(* Logix 5000 project; controller Modbus_TCP_Client_Example vendor 1 type 14 code 154 rev 32.15; software revision 32.05 *)

TASK Modbus_Task (periodic, rate 50 ms, priority 10, watchdog 500 ms) : Modbus_Program   // Conveyor MDXT

MODULES
   Local : vendor 1 type 14 code 154 (PointIO 0, rev 32.15)
      Discrete_IO : Embedded (PointIO 1, rev 32.11, Output RPI 20 ms)
END_MODULES

TYPE AMP_Alarm_Word :   // Applied Motion Input Assembly - Alarm Word
STRUCT
   Position_Limit : BOOL;   // Position Limit
   CCW_Limit : BOOL;   // CCW Limit
   CW_Limit : BOOL;   // CW Limit
   Over_Temp : BOOL;   // Over Temp
   Excess_Regen_or_Internal_Voltage : BOOL;   // Excess Regen or Internal Voltage
   Over_Voltage : BOOL;   // Over Voltage
   Under_Voltage : BOOL;   // Under Voltage
   Over_Current : BOOL;   // Over Current
   Open_Motor_Windings : BOOL;   // Open Motor Windings
   Bad_Encoder : BOOL;   // Bad Encoder
   Comm_Error : BOOL;   // Comm Error
   Bad_Flash : BOOL;   // Bad Flash
   No_Move : BOOL;   // No Move
   NA_1 : BOOL;   // NA 1
   Blank_Q_Segment : BOOL;   // Blank Q Segment
   NA_2 : BOOL;   // NA 2
END_STRUCT
END_TYPE

TYPE AMP_Input_Assembly_Servo_v2 :   // Applied Motion Servo Drive Input Assembly Version 1.0
STRUCT
   Control_Word_Received : DINT;   // Control Word Status equals to Control Words sent in Output Assembly
   OpCode1_Received : DINT;   // OpCode 1 Status equals to OpCode1 sent in Output Assembly
   Control_Mode : DINT;   // Control Mode Status: Position, Torque, Gear
   Status_Code : DINT;   // Status Code
   Alarm_Code : DINT;   // Alarm Code
   Supply_Voltage : DINT;   // Supply Voltage 0.1 V: ex. 242=24.2V
   Applied_Torque : DINT;   // Total Applied Torque %
   Drive_Temperature : DINT;   // Drive Temperature 0.1 deg C: ex. 305=30.5 C
   Encoder_Position : DINT;   // Encoder Position
   Second_Encoder_Position : DINT;   // Absolute Position
   Position_Error : DINT;   // Position Error in Counts
   Actual_Velocity_RPS : DINT;   // Actual Velocity rev/sec*2: ex. 480=2 rev/sec
   Digital_Outputs : DINT;   // Digital Output Status
   Digital_Inputs : DINT;   // Digital Input Status
   Analog_Output1 : DINT;   // 0 = min V, 16383 = max V
   Analog_Output2 : DINT;   // 0 = min V, 16383 = max V
   Analog_Input1 : DINT;   // 0 = min V, 16383 = max V
   Analog_Input2 : DINT;   // 0 = min V, 16383 = max V
   Torque_Limit : DINT;   // Torque Limit Set Point Feedback
   Second_Encoder_Speed : DINT;   // External Encoder Speed Feedback if any
END_STRUCT
END_TYPE

TYPE AMP_Input_Assembly_v2 :   // Applied Motion Drive Input Assembly Version 2.0
STRUCT
   Status_Code : DINT;   // Status Code
   Alarm_Code : DINT;   // Alarm Code
   Voltage : DINT;   // Supply Voltage (x0.1V)
   Current : DINT;   // Actual Current (mA)
   Temp : DINT;   // Drive Temperature (0.1 deg C)
   Encoder_Position : DINT;   // Encoder Position (20,000 counts = 1 shaft turn)
   Absolute_Position : DINT;   // Absolute Position (20,000 counts = 1 shaft turn)
   Position_Error : DINT;   // Position Error (counts)
   Actual_Velocity : DINT;   // Actual Velocity (rev/sec * 240, 0 when no encoder)
   Extended_Inputs : DINT;   // Input Status (Extended)
   Main_Board_Inputs : DINT;   // Input Status (Main board)
   Word11 : DINT;   // Reserved
   Analog_Input_1 : DINT;   // Analog Input 1 (ADC counts, 0=min V, 16383 = max V)
   Analog_Input_2 : DINT;   // Analog Input 2 (ADC counts, 0=min V, 16383 = max V)
END_STRUCT
END_TYPE

TYPE AMP_Status_Word :   // Applied Motion Input Assembly Status Word
STRUCT
   Enabled : BOOL;   // Motor Enabled (Motor Disabled if this bit = 0)
   Sampling : BOOL;   // Sampling (for Quick Tuner)
   Drive_Fault : BOOL;   // Drive Fault (check Alarm Code)
   In_Position : BOOL;   // In Position (motor is in position)
   Moving : BOOL;   // Moving (motor is moving)
   Jogging : BOOL;   // Jogging (currently in jog mode)
   Stopping : BOOL;   // Stopping (in the process of stopping from a stop command)
   Waiting : BOOL;   // Waiting (for an input; executing a WI command)
   Saving : BOOL;   // Saving (parameter data is being saved)
   Alarm_Present : BOOL;   // Alarm present (check Alarm Code)
   Homing : BOOL;   // Homing (executing an SH command)
   Wait_Time : BOOL;   // Waiting (for time; executing a WD or WT command)
   Wizard_Running : BOOL;   // Wizard running (Timing Wizard is running)
   Checking_Encoder : BOOL;   // Checking encoder (Timing Wizard is running)
   Q_Program_Running : BOOL;   // Q Program is running
   Initializing : BOOL;   // Initializing (happens at power up) ; Servo Ready (for SV200 drives only)
END_STRUCT
END_TYPE

TYPE AMP_Status_Word_Servo :   // Applied Motion Input Assembly Status Word 'SC'
STRUCT
   Enabled : BOOL;   // Motor Enabled (Motor Disabled if this bit = 0)
   Sampling : BOOL;   // Sampling
   Drive_Fault : BOOL;   // Drive Fault (check Alarm Code)
   In_Position : BOOL;   // In Position (motor is in position)
   Moving : BOOL;   // Moving (motor is moving)
   Jogging : BOOL;   // Jogging (currently in jog mode)
   Stopping : BOOL;   // Stopping (in the process of stopping from a stop command)
   Waiting : BOOL;   // Waiting (for an input; executing a WI command)
   Saving : BOOL;   // Saving (parameter data is being saved)
   Alarm_Present : BOOL;   // Alarm present (check Alarm Code)
   Homing : BOOL;   // Homing (executing an SH command)
   Wait_Time : BOOL;   // Waiting (for time; executing a WD or WT command)
   Wizard_Running : BOOL;   // Wizard running (Timing Wizard is running)
   Checking_Encoder : BOOL;   // Checking encoder (Timing Wizard is running)
   Q_Program_Running : BOOL;   // Q Program is running
   Servo_Ready : BOOL;   // Servo Ready;Initializing (happens at power up)
   CSP_Following : BOOL;
   In_Velocity : BOOL;   // Velocity Reached
   Zero_Speed : BOOL;   // Motor is standstill
   Torque_Reached : BOOL;   // Toruqe Target Reached
   In_Torque : BOOL;   // Current Control Mode is Torque
   Group2_PID : BOOL;   // The Second Set of Gain is Valid
   Secondary_Control_Mode : BOOL;   // Second Control Mode is in Operation
   Velocity_Reached : BOOL;   // Velocity Target Reached
   Homing_Complete : BOOL;   // Homing Completed Feedback
END_STRUCT
END_TYPE

TYPE raC_UDT_ModbusClientConnection :
STRUCT
   LocalSlot : SINT;   // Local Slot for Ethernet module. For ControlLogix - L8x, EN2T(R) - use the actual module slot. For CompactLogix use slot 0.
   LocalAddress : STR0016;   // Used only for controllers with more than 1 local IP address (5380, 5480). For all others must be blank.
   DestAddress : STR0016;   // The IP address for the Modbus TCP Slave device to connect to
   DestinationPort : DINT;   // Default Modbus is 502
   MSG_Src : SINT[500];   // Placeholder for message source
   MSG_Dest : SINT[500];   // Placeholder for message destination
END_STRUCT
END_TYPE

TYPE raC_UDT_ModbusClientData :
STRUCT
   Coils_0xxx : BOOL[1024];
   DiscInputs_1xxx : BOOL[1024];
   InpRegisters_3xxx : INT[1024];
   HoldRegisters_4xxx : INT[1024];
END_STRUCT
END_TYPE

TYPE raC_UDT_ModbusClientHMI :
STRUCT
   Parameters : raC_UDT_ModbusClientConnection;
   Transaction : raC_UDT_ModbusClientTransaction;
   Index0x : DINT;
   Index1x : DINT;
   Index3x : DINT;
   Index4x : DINT;
   DataValue : INT[65];
   DataAddr : DINT[65];
   TransactionIndex : DINT;
   RemoteAddrStart : DINT;
   RemoteAddrEnd : DINT;
   LocalAddrEnd : DINT;
END_STRUCT
END_TYPE

TYPE raC_UDT_ModbusClientTransaction :
STRUCT
   Enabled : BOOL;   // Enables (1) or disables (0) the transaction
   PollInterval : DINT;   // Time between triggers in milliseconds. Minimum is 80 msec. Anyting below 80 will be set to 1 seconds
   TransType : INT;   // Transaction code for the Modbus Protocol. Acceptable values are 1-Coil Read, 2- Discrete Input read, 3-Holding Register Read, 4-Input Register Read, 5-Write Single Coil, 6-Single Holding Register Write, 15-Multiple Coil Write, 16 Multiple Holding Register Write
   StationID : SINT;   // Station ID ( Unit Identifier). Commonly used if going through a gateway or bridge in which case it is the device address on the other side of the gateway. Other wise leave as 0
   BeginAddress : DINT;   // Beginning address in remote device to read from or write to.
   Count : INT;   // The number of items in remote device to read from or write to.
   LocalAddress : INT;   // Beginning address in in this programs' "_Data" arrays
   TransComplete : BOOL;   // Transaction Complete Flag. Check the TransStat to see if the transaction was successful or if a Modbus exception code was returned.
   TransStat : INT;   // Status result of the transaction. 0 = success, 1 = in process 2 = retry -1 = exception
   Diagnostic : raC_UDT_ModbusClientTransactionDiag;
END_STRUCT
END_TYPE

TYPE raC_UDT_ModbusClientTransactionDiag :
STRUCT
   Request : STR0500;   // Actual buffer used to build the modbus request that is transmited to the remote node.
   ReqBuilt : BOOL;   // Transaction request string is built, clear this if anything is changed in a read operation to rebuild the Request string.
   Overlap : BOOL;   // Transaction is not completing before next trigger
   Overload : BOOL;   // Transaction is not completing because of excessive Overlaps in one or more transactions
   TransID : INT;   // Serial Number of the actual Ethernet Transaction used to match to the appropriate Reply
   TransLastError : INT;   // Last Error on transaction. 0-Success, -2 Network write error, -3 Local write error, -4 Network Read Error, -5 Local Read Error, -6 Connection failed.. -12 Invalid Trans code, -13 Out of data array range.
   IntervalTimer : TIMER;   // IntervalTimer, used to trigger transaction
   NoReplyCounter : COUNTER;   // No Reply Counter
   PendingTimer : TIMER;   // Timing pending requests
END_STRUCT
END_TYPE

TYPE raC_UDT_ModbusConnectParam :   // Parameterss for the OpenConnection Service
STRUCT
   Timeout : DINT;
   DestAddr : STR0032;
END_STRUCT
END_TYPE

TYPE raC_UDT_ModbusCreateParam :
STRUCT
   Type : DINT;   // Type 1-TCP, 2-UDP
   Family : INT;   // Address Family Must be 2
   Port : INT;   // Local Port Number
   Addr : DINT;   // Local IP Address
END_STRUCT
END_TYPE

TYPE STR0008 :
STRUCT
   LEN : DINT;
   DATA : SINT[8];
END_STRUCT
END_TYPE

TYPE STR0016 :
STRUCT
   LEN : DINT;
   DATA : SINT[16];
END_STRUCT
END_TYPE

TYPE STR0032 :
STRUCT
   LEN : DINT;
   DATA : SINT[32];
END_STRUCT
END_TYPE

TYPE STR0500 :
STRUCT
   LEN : DINT;
   DATA : SINT[500];
END_STRUCT
END_TYPE

TYPE STR4096 :
STRUCT
   LEN : DINT;
   DATA : SINT[4096];
END_STRUCT
END_TYPE

ADD_ON_INSTRUCTION AMP_Absolute_Move   (* revision 1.0 *)
// Applied Motion - Absolute Move AOI
// Help:
// The Absolute Move AOI is used to move an axis to a specified absolute position.
VAR_IN_OUT
   Input : DINT[14]; {required}   // Drive Input Assembly
   Output : DINT[16]; {required}   // Drive Output Assembly
        [0]   // Command Word
        [10]   // Data/Register 1
        [11]   // Data/Register 2
        [1]   // Jog Speed (0.25 rev/min)
        [2]   // Jog Acceleration (10 rev/s/s)
        [3]   // Jog Deceleration (10 rev/s/s)
        [4]   // Point-to-Point Velocity (0.25 rev/min)
        [5]   // Point-to-Point Acceleration (10 rev/min/s)
        [6]   // Point-to-Point Deceleration (10 rev/min/s)
        [7]   // Point-to-Point Distance (Motor steps)
        [9]   // (2x ASCII Letters in 16 lower word)
END_VAR
VAR_INPUT
   RPI : DINT := 100; {visible}   // Drive Connection Request Packet Interval (milliseconds)
   Start : BOOL; {required}   // Start the Relative Move
   Position : DINT; {required}   // Destination Position (steps, negative = reverse)
   Speed : REAL; {required}   // Velocity of Move (rev/min)
   Acc : REAL; {required}   // Acceleration of Move (rev/s/s)
   Dec : REAL; {required}   // Deceleration (rev/s/s)
END_VAR
VAR_OUTPUT
   Sent : BOOL; {access Read Only, visible}   // Move has been sent to drive
   In_Progress : BOOL; {access Read Only, visible}   // Move in progress
   Done : BOOL; {access Read Only, visible}   // Move completed without errors - desired position reached
   Error : BOOL; {access Read Only, visible}   // Move failed to complete - drive not ready or faulted
   State : DINT := 10; {access Read Only}   // Internal state of progress
END_VAR
VAR
   Loc_StatusCode : AMP_Status_Word;
   Loc_CommandOff_Timer : TIMER;   // Timer to make sure command value was 0 before sending a new command
   Loc_CommandOn_Timer : TIMER;   // Timer to make sure command value is set long enough to be sent to drive
   Loc_Input_Assembly : AMP_Input_Assembly_v2; {access None}
   Loc_Start_ONS : BOOL; {access None}
   Loc_AlarmCode : AMP_Alarm_Word; {access None}
END_VAR

ROUTINE Logic   (* ladder *)
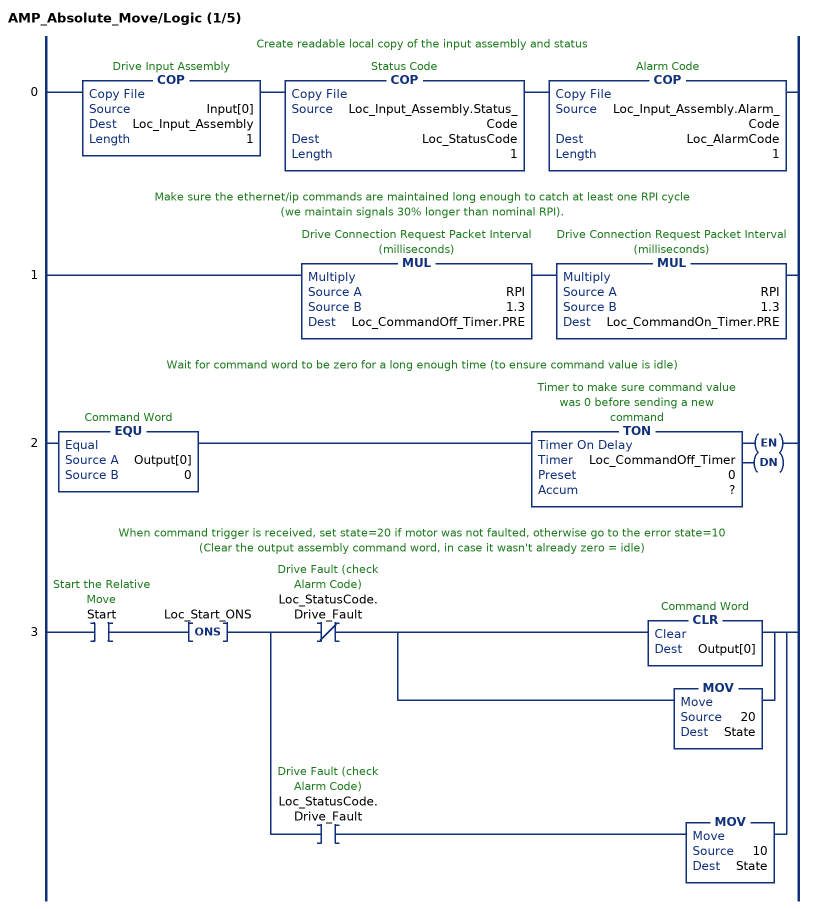
   // Create readable local copy of the input assembly and status
   0: COP(Input[0],Loc_Input_Assembly,1)COP(Loc_Input_Assembly.Status_Code,Loc_StatusCode,1)COP(Loc_Input_Assembly.Alarm_Code,Loc_AlarmCode,1);
   // Make sure the ethernet/ip commands are maintained long enough to catch at least one RPI cycle
   // (we maintain signals 30% longer than nominal RPI).
   1: MUL(RPI,1.3,Loc_CommandOff_Timer.PRE)MUL(RPI,1.3,Loc_CommandOn_Timer.PRE);
   // Wait for command word to be zero for a long enough time (to ensure command value is idle)
   2: EQU(Output[0],0)TON(Loc_CommandOff_Timer,?,?);
   // When command trigger is received, set state=20 if motor was not faulted, otherwise go to the error state=10
   // (Clear the output assembly command word, in case it wasn't already zero = idle)
   3: XIC(Start)ONS(Loc_Start_ONS)[XIO(Loc_StatusCode.Drive_Fault) [CLR(Output[0]) ,MOV(20,State) ] ,XIC(Loc_StatusCode.Drive_Fault) MOV(10,State) ];
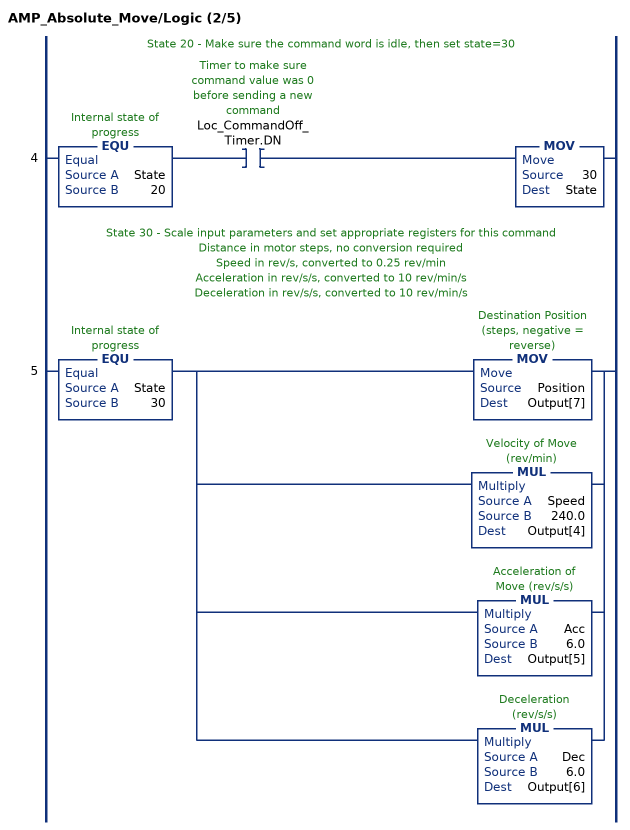
   // State 20 - Make sure the command word is idle, then set state=30
   4: EQU(State,20)XIC(Loc_CommandOff_Timer.DN)MOV(30,State);
   // State 30 - Scale input parameters and set appropriate registers for this command
   // Distance in motor steps, no conversion required
   // Speed in rev/s, converted to 0.25 rev/min
   // Acceleration in rev/s/s, converted to 10 rev/min/s
   // Deceleration in rev/s/s, converted to 10 rev/min/s
   5: EQU(State,30)[MOV(Position,Output[7]) ,MUL(Speed,240.0,Output[4]) ,MUL(Acc,6.0,Output[5]) ,MUL(Dec,6.0,Output[6]) ];
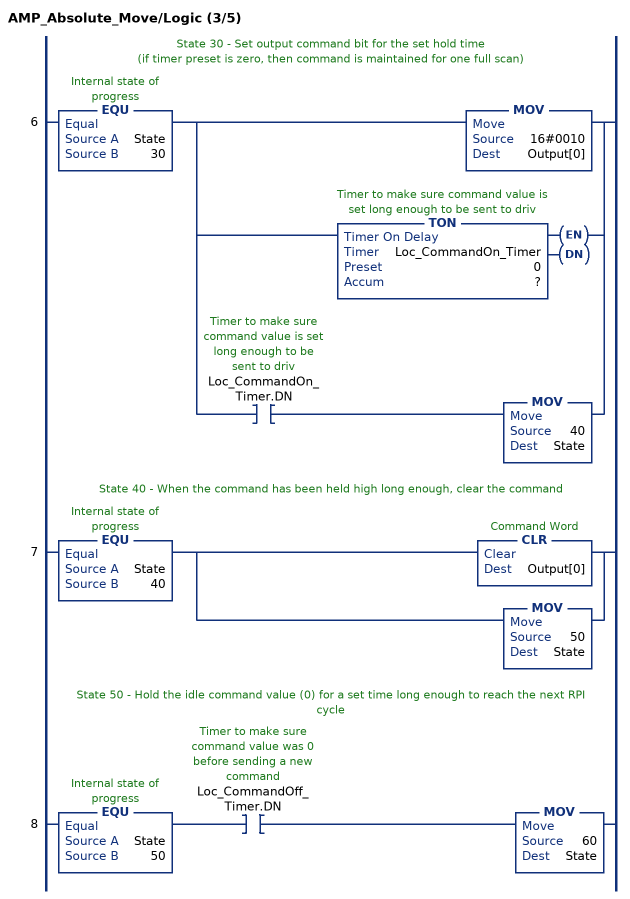
   // State 30 - Set output command bit for the set hold time
   // (if timer preset is zero, then command is maintained for one full scan)
   6: EQU(State,30)[MOV(16#0010,Output[0]) ,TON(Loc_CommandOn_Timer,?,?) ,XIC(Loc_CommandOn_Timer.DN) MOV(40,State) ];
   // State 40 - When the command has been held high long enough, clear the command
   7: EQU(State,40)[CLR(Output[0]) ,MOV(50,State) ];
   // State 50 - Hold the idle command value (0) for a set time long enough to reach the next RPI cycle
   8: EQU(State,50)XIC(Loc_CommandOff_Timer.DN)MOV(60,State);
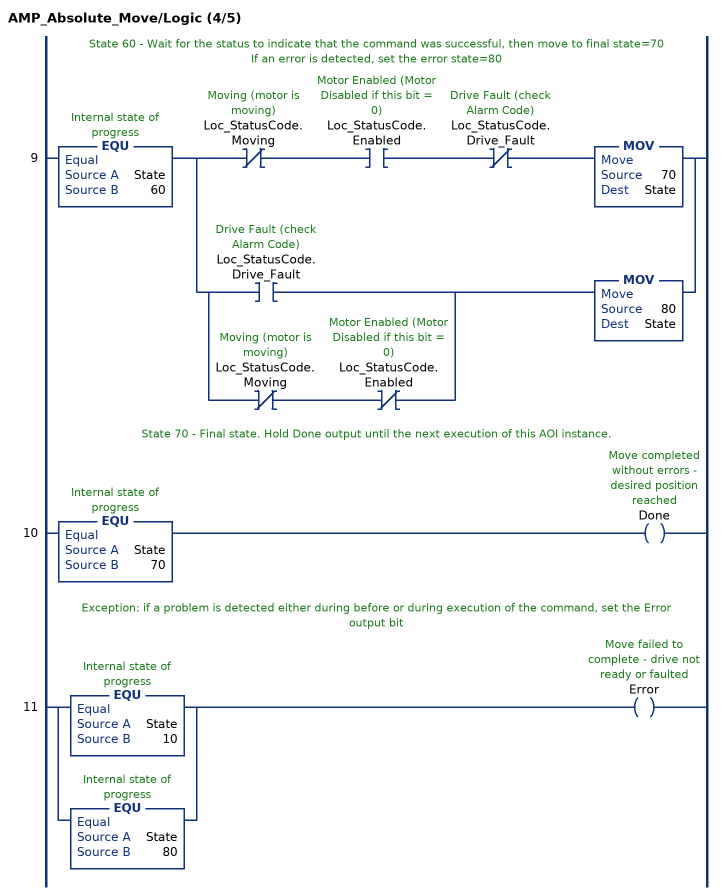
   // State 60 - Wait for the status to indicate that the command was successful, then move to final state=70
   // If an error is detected, set the error state=80
   9: EQU(State,60)[XIO(Loc_StatusCode.Moving) XIC(Loc_StatusCode.Enabled) XIO(Loc_StatusCode.Drive_Fault) MOV(70,State) ,[XIC(Loc_StatusCode.Drive_Fault) ,XIO(Loc_StatusCode.Moving) XIO(Loc_StatusCode.Enabled) ] MOV(80,State) ];
   // State 70 - Final state. Hold Done output until the next execution of this AOI instance.
   10: EQU(State,70)OTE(Done);
   // Exception: if a problem is detected either during before or during execution of the command, set the Error output bit
   11: [EQU(State,10) ,EQU(State,80) ]OTE(Error);
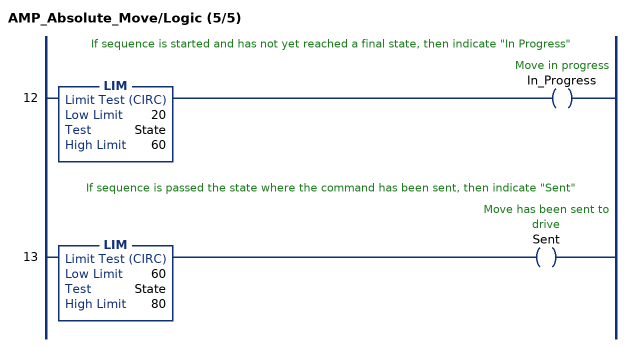
   // If sequence is started and has not yet reached a final state, then indicate "In Progress"
   12: LIM(20,State,60)OTE(In_Progress);
   // If sequence is passed the state where the command has been sent, then indicate "Sent"
   13: LIM(60,State,80)OTE(Sent);
END_ROUTINE
END_ADD_ON_INSTRUCTION

ADD_ON_INSTRUCTION AMP_Absolute_Move_Servo   (* revision 1.0, vendor Applied Motion Products Inc. *)
// Applied Motion - Motor Absolute Move - AOI
// Help:
// The Absolute Move AOI is used to move an axis to a specified absolute position(FP).
VAR_IN_OUT
   Input : DINT[20]; {required}   // Drive Input Assembly
        [16]   // Analog_Input1
        [4]   // Alarm_Code
        [0]   // Control_Word_Received
        [10]   // Position_Error
        [11]   // Actual_Velocity_RPS
        [12]   // Digital_Outputs
        [13]   // Digital_Inputs
        [14]   // Analog_Output1
        [15]   // Analog_Output2
        [17]   // Analog_Input2
        [18]   // Torque_Limit
        [19]   // Second_Encoder_Speed
        [1]   // OpCode1_Received
        [2]   // Control_Mode
        [3]   // Status_Code
        [5]   // Supply_Voltage
        [6]   // Applied_Torque
        [7]   // Drive_Temperature
        [8]   // Encoder_Position
        [9]   // Second_Encoder_Position
   Output : DINT[11]; {required}   // Drive Output Assembly
        [10]   // Reserved
        [4]   // Target Velocity
        [0]   // Control Word
        [3]   // Target Pos
        [1]   // OpCode 1
        [2]   // OpCode 2
        [5]   // Porifle Acceleration
        [6]   // Profile Deceleration
        [7]   // Target Torque
        [8]   // OpCode 3
        [9]   // OpCode 4
END_VAR
VAR_INPUT
   Start : BOOL; {required}   // Start the Absolute Move
   Position : DINT; {required}   // Destination Position (negative = reverse)
   Speed_rps : REAL; {required}   // Velocity of Move (rev/sec)
   Acc : REAL; {required}   // Acceleration of Move (rev/s/s)
   Dec : REAL; {required}   // Deceleration of Move (rev/s/s)
END_VAR
VAR_OUTPUT
   Sent : BOOL; {access Read Only, visible}   // Move has been sent to drive
   In_Progress : BOOL; {access Read Only, visible}   // Move in progress
   Done : BOOL; {access Read Only, visible}   // Move completed without errors - desired position reached
   Error : BOOL; {access Read Only, visible}   // Move failed to complete - drive not ready or faulted
   State : DINT := 10; {access Read Only}   // Internal state of progress
END_VAR
VAR
   Loc_StatusCode : AMP_Status_Word_Servo; {access None}
   Loc_Input_Assembly : AMP_Input_Assembly_Servo_v2; {access None}
   Loc_Abs_ONS : BOOL;
   Loc_Command_Timeout : TIMER := (PRE := 2000); {access None}   // Timer to output fault if command is not Done
END_VAR

ROUTINE Logic   (* ladder *)
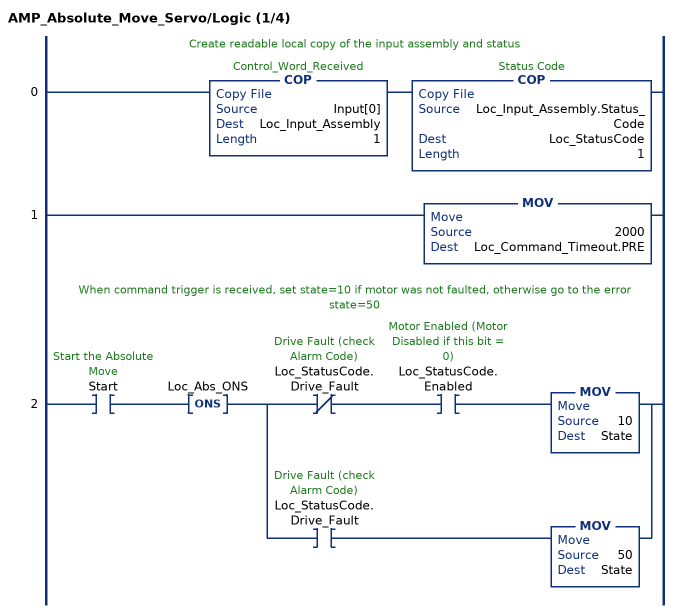
   // Create readable local copy of the input assembly and status
   0: COP(Input[0],Loc_Input_Assembly,1)COP(Loc_Input_Assembly.Status_Code,Loc_StatusCode,1);
   1: MOV(2000,Loc_Command_Timeout.PRE);
   // When command trigger is received, set state=10 if motor was not faulted, otherwise go to the error state=50
   2: XIC(Start)ONS(Loc_Abs_ONS)[XIO(Loc_StatusCode.Drive_Fault) XIC(Loc_StatusCode.Enabled) MOV(10,State) ,XIC(Loc_StatusCode.Drive_Fault) MOV(50,State) ];
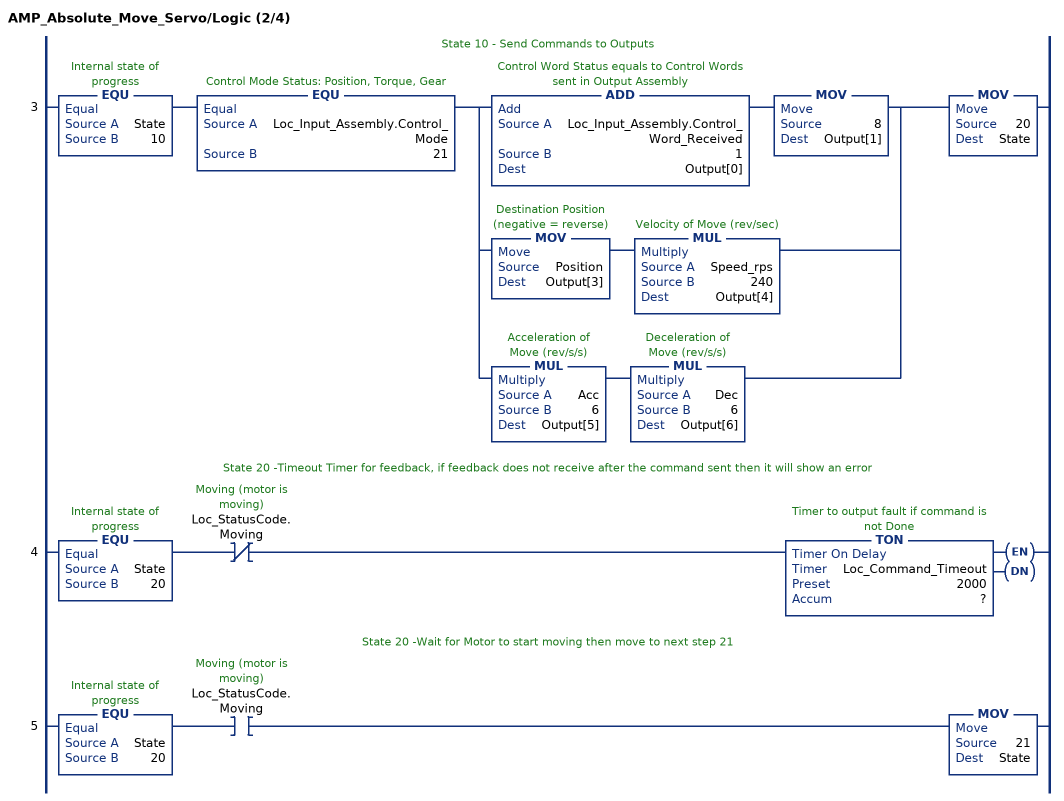
   // State 10 - Send Commands to Outputs
   3: EQU(State,10)EQU(Loc_Input_Assembly.Control_Mode,21)[ADD(Loc_Input_Assembly.Control_Word_Received,1,Output[0]) MOV(8,Output[1]) ,MOV(Position,Output[3]) MUL(Speed_rps,240,Output[4]) ,MUL(Acc,6,Output[5]) MUL(Dec,6,Output[6]) ]MOV(20,State);
   // State 20 -Timeout Timer for feedback, if feedback does not receive after the command sent then it will show an error
   4: EQU(State,20)XIO(Loc_StatusCode.Moving)TON(Loc_Command_Timeout,?,?);
   // State 20 -Wait for Motor to start moving then move to next step 21
   5: EQU(State,20)XIC(Loc_StatusCode.Moving)MOV(21,State);
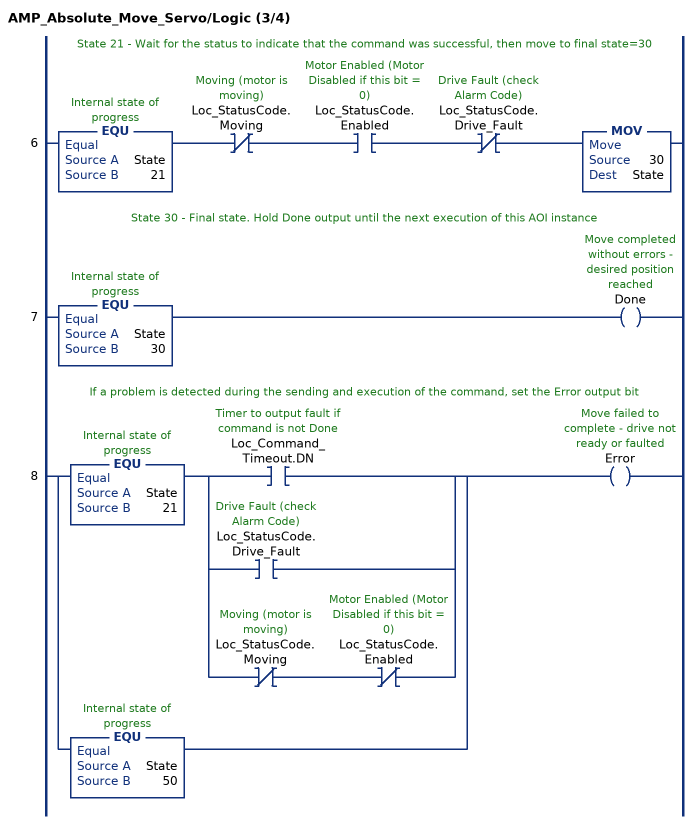
   // State 21 - Wait for the status to indicate that the command was successful, then move to final state=30
   6: EQU(State,21)XIO(Loc_StatusCode.Moving)XIC(Loc_StatusCode.Enabled)XIO(Loc_StatusCode.Drive_Fault)MOV(30,State);
   // State 30 - Final state. Hold Done output until the next execution of this AOI instance
   7: EQU(State,30)OTE(Done);
   // If a problem is detected during the sending and execution of the command, set the Error output bit
   8: [EQU(State,21) [XIC(Loc_Command_Timeout.DN) ,XIC(Loc_StatusCode.Drive_Fault) ,XIO(Loc_StatusCode.Moving) XIO(Loc_StatusCode.Enabled) ] ,EQU(State,50) ]OTE(Error);
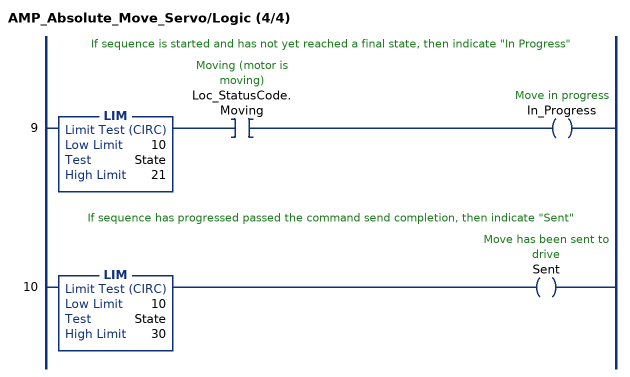
   // If sequence is started and has not yet reached a final state, then indicate "In Progress"
   9: LIM(10,State,21)XIC(Loc_StatusCode.Moving)OTE(In_Progress);
   // If sequence has progressed passed the command send completion, then indicate "Sent"
   10: LIM(10,State,30)OTE(Sent);
END_ROUTINE
END_ADD_ON_INSTRUCTION

ADD_ON_INSTRUCTION AMP_Alarm_Code   (* revision 1.0 *)
// Applied Motion - Alarm Code - AOI
// Help:
// The Alarm Code AOI uses the raw data stored in the Alarm Code word (Element 1 from Input Assembly 0x65) to set individual appropriately named boolean outputs.
VAR_INPUT
   Input : DINT; {required}   // Element 1 from Drive Input Assembly (0x65)
END_VAR
VAR_OUTPUT
   Position_Limit : BOOL; {access Read Only, visible}
   CCW_Limit : BOOL; {access Read Only, visible}
   CW_Limit : BOOL; {access Read Only, visible}
   Over_Temp : BOOL; {access Read Only, visible}
   Excess_Regen_or_Internal_Voltage : BOOL; {access Read Only, visible}
   Over_Voltage : BOOL; {access Read Only, visible}
   Under_Voltage : BOOL; {access Read Only, visible}
   Over_Current : BOOL; {access Read Only, visible}
   Open_Motor_Windings : BOOL; {access Read Only, visible}
   Bad_Encoder : BOOL; {access Read Only, visible}
   Comm_Error : BOOL; {access Read Only, visible}
   Bad_Flash : BOOL; {access Read Only, visible}
   No_Move : BOOL; {access Read Only, visible}
   NA_1 : BOOL; {access Read Only, visible}
   Blank_Q_Segment : BOOL; {access Read Only, visible}
   NA_2 : BOOL; {access Read Only, visible}
END_VAR

ROUTINE Logic   (* ladder *)
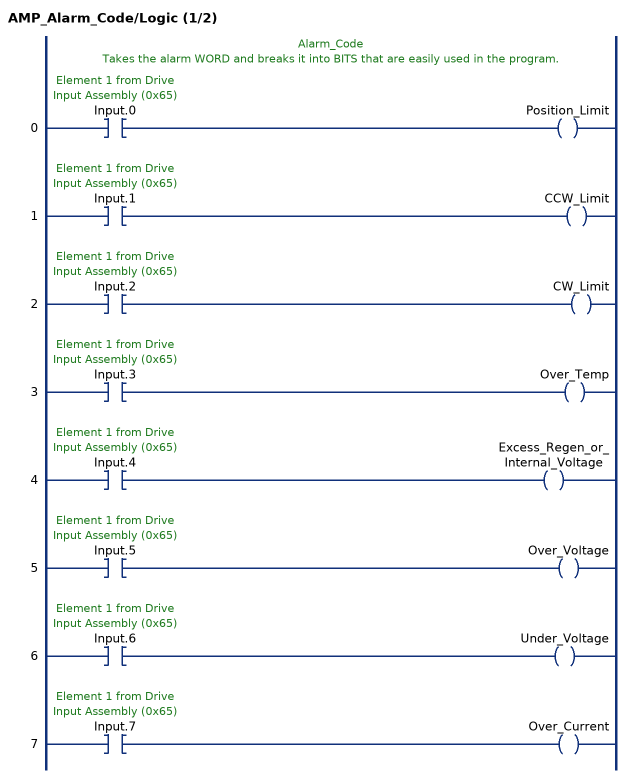
   // Alarm_Code
   // Takes the alarm WORD and breaks it into BITS that are easily used in the program.
   0: XIC(Input.0)OTE(Position_Limit);
   1: XIC(Input.1)OTE(CCW_Limit);
   2: XIC(Input.2)OTE(CW_Limit);
   3: XIC(Input.3)OTE(Over_Temp);
   4: XIC(Input.4)OTE(Excess_Regen_or_Internal_Voltage);
   5: XIC(Input.5)OTE(Over_Voltage);
   6: XIC(Input.6)OTE(Under_Voltage);
   7: XIC(Input.7)OTE(Over_Current);
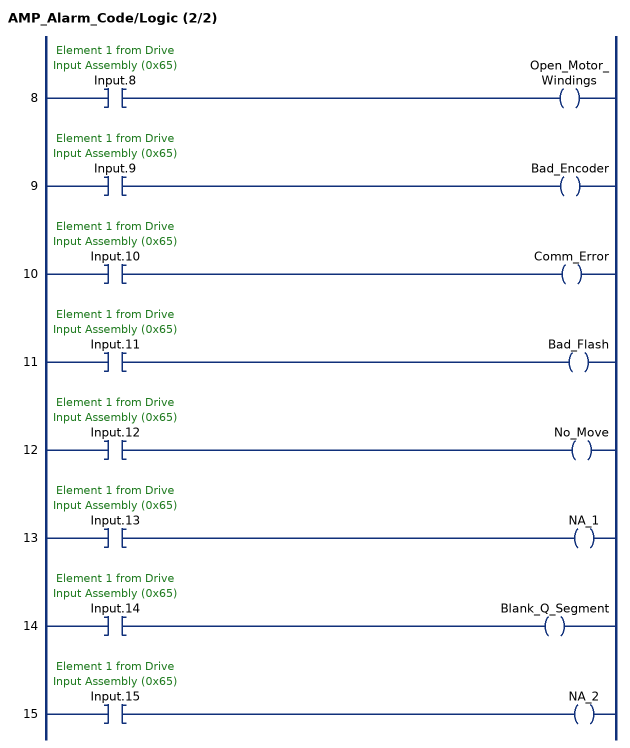
   8: XIC(Input.8)OTE(Open_Motor_Windings);
   9: XIC(Input.9)OTE(Bad_Encoder);
   10: XIC(Input.10)OTE(Comm_Error);
   11: XIC(Input.11)OTE(Bad_Flash);
   12: XIC(Input.12)OTE(No_Move);
   13: XIC(Input.13)OTE(NA_1);
   14: XIC(Input.14)OTE(Blank_Q_Segment);
   15: XIC(Input.15)OTE(NA_2);
END_ROUTINE
END_ADD_ON_INSTRUCTION

ADD_ON_INSTRUCTION AMP_Alarm_Code_Servo   (* revision 1.0, vendor Applied Motion Products Inc. *)
// Applied Motion - Alarm Code(AL) AOI
// Help:
// The Alarm Code AOI uses the raw data stored in the Alarm Code word (Element 1 from Input Assembly) to set individual appropriately named boolean outputs.
VAR_INPUT
   Input : DINT; {access Read Only, required}   // Element 5 from Drive Input Assembly
END_VAR
VAR_OUTPUT
   Over_Temp_Fault : BOOL; {access Read Only, visible}   // Over temperature error
   Position_Error_Fault : BOOL; {access Read Only, visible}   // Position Error Limit Fault
   Internal_Error_Fault : BOOL; {access Read Only, visible}   // Internal error fault
   Out_of_Range_Voltage_Fault : BOOL; {access Read Only, visible}   // Power voltage over range
   Over_Current_Fault : BOOL; {access Read Only, visible}   // Over current occured
   Safety_Torque_Off_Fault : BOOL; {access Read Only, visible}   // STO fault occured
   Encoder_Disconnected_Fault : BOOL; {access Read Only, visible}   // Encoder is disconnected
   Velocity_Exceed_Limit_Fault : BOOL; {access Read Only, visible}   // Velocity limit fault
   Abnormal_Motion_Protection_Fault : BOOL; {access Read Only, visible}   // Abnormal motion protection fault
   EthernetIP_Comm_Fault : BOOL; {access Read Only, visible}   // Communication error
   Hybrid_Deviation_Fault : BOOL; {access Read Only, visible}   // Hybrid deviation error fault (full closed loop operationl)
   Secondary_Encoder_Disconnected_Fault : BOOL; {access Read Only, visible}   // Secondary Encoder is not connected (full closed loop operation)
   Emergenecy_Stop_Warning : BOOL; {access Read Only, visible}   // Emergency stop is on
   Regen_Failed_Warning : BOOL; {access Read Only, visible}   // Regen failed warning
   CCW_Limit_Warning : BOOL; {access Read Only, visible}   // Counterclockwise limit
   CW_Limit_Warning : BOOL; {access Read Only, visible}   // Clockwise limit
   Peak_Current_Foldback_Warning : BOOL; {access Read Only, visible}   // Peak Current CP foldback error
   Abnormal_StartUp_Warning : BOOL; {access Read Only, visible}   // Abnormal Start of the motor
   Abnormal_Communication_Warning : BOOL; {access Read Only, visible}   // Abnormal Communication
   Under_Voltage_Warning : BOOL; {access Read Only, visible}   // Undervoltage supply error
   Absolute_Position_Lost_Warning : BOOL; {access Read Only, visible}   // Absolute position lost error
   Absolute_Position_Overflow_Warning : BOOL; {access Read Only, visible}   // Absolute position overflow error
   Absolute_Postion_MultiTurn_Warning : BOOL; {access Read Only, visible}   // Absolute multiturn error
   Homing_Parameter_Warning : BOOL; {access Read Only, visible}   // Wrong homing parameter entered
   Phase_Lost_Warning : BOOL; {access Read Only, visible}   // Motor main power phase lost
   Absolute_Battery_Encoder_Voltage_Warning : BOOL; {access Read Only, visible}   // Absolute Encoder battey is under voltage
   Reserved : INT; {access Read Only}
END_VAR

ROUTINE Logic   (* ladder *)
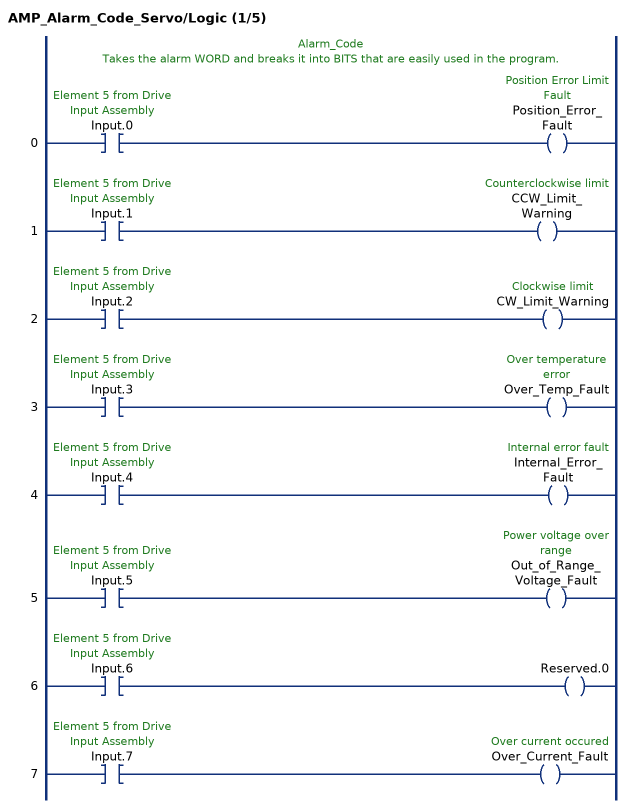
   // Alarm_Code
   // Takes the alarm WORD and breaks it into BITS that are easily used in the program.
   0: XIC(Input.0)OTE(Position_Error_Fault);
   1: XIC(Input.1)OTE(CCW_Limit_Warning);
   2: XIC(Input.2)OTE(CW_Limit_Warning);
   3: XIC(Input.3)OTE(Over_Temp_Fault);
   4: XIC(Input.4)OTE(Internal_Error_Fault);
   5: XIC(Input.5)OTE(Out_of_Range_Voltage_Fault);
   6: XIC(Input.6)OTE(Reserved.0);
   7: XIC(Input.7)OTE(Over_Current_Fault);
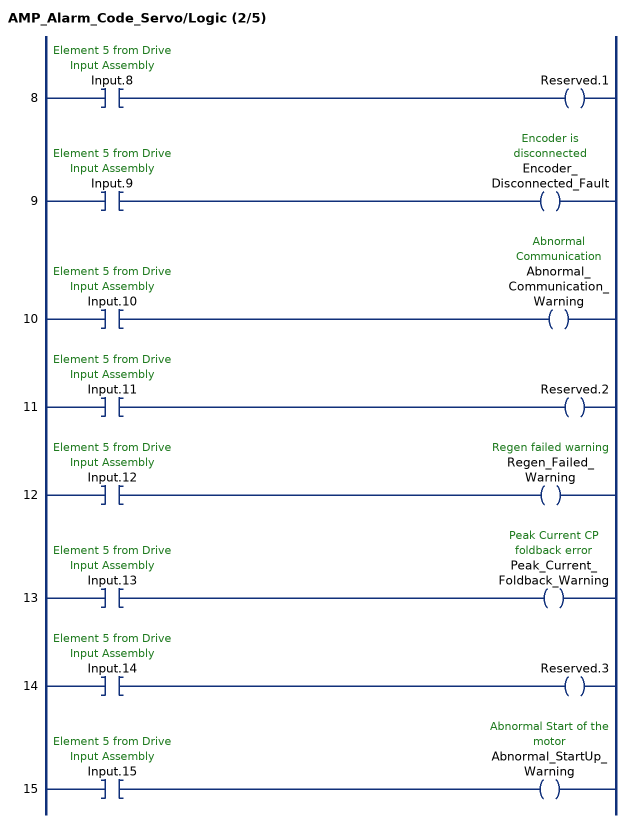
   8: XIC(Input.8)OTE(Reserved.1);
   9: XIC(Input.9)OTE(Encoder_Disconnected_Fault);
   10: XIC(Input.10)OTE(Abnormal_Communication_Warning);
   11: XIC(Input.11)OTE(Reserved.2);
   12: XIC(Input.12)OTE(Regen_Failed_Warning);
   13: XIC(Input.13)OTE(Peak_Current_Foldback_Warning);
   14: XIC(Input.14)OTE(Reserved.3);
   15: XIC(Input.15)OTE(Abnormal_StartUp_Warning);
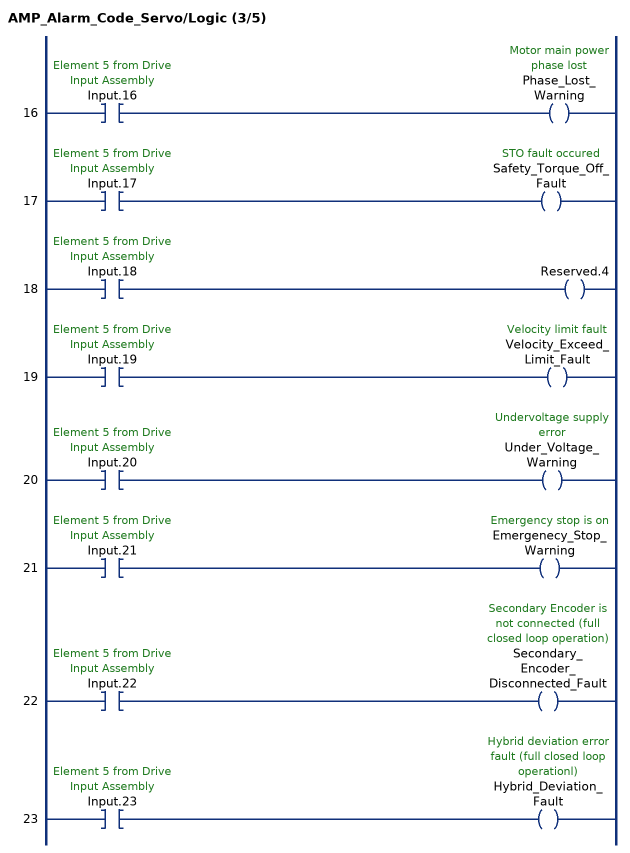
   16: XIC(Input.16)OTE(Phase_Lost_Warning);
   17: XIC(Input.17)OTE(Safety_Torque_Off_Fault);
   18: XIC(Input.18)OTE(Reserved.4);
   19: XIC(Input.19)OTE(Velocity_Exceed_Limit_Fault);
   20: XIC(Input.20)OTE(Under_Voltage_Warning);
   21: XIC(Input.21)OTE(Emergenecy_Stop_Warning);
   22: XIC(Input.22)OTE(Secondary_Encoder_Disconnected_Fault);
   23: XIC(Input.23)OTE(Hybrid_Deviation_Fault);
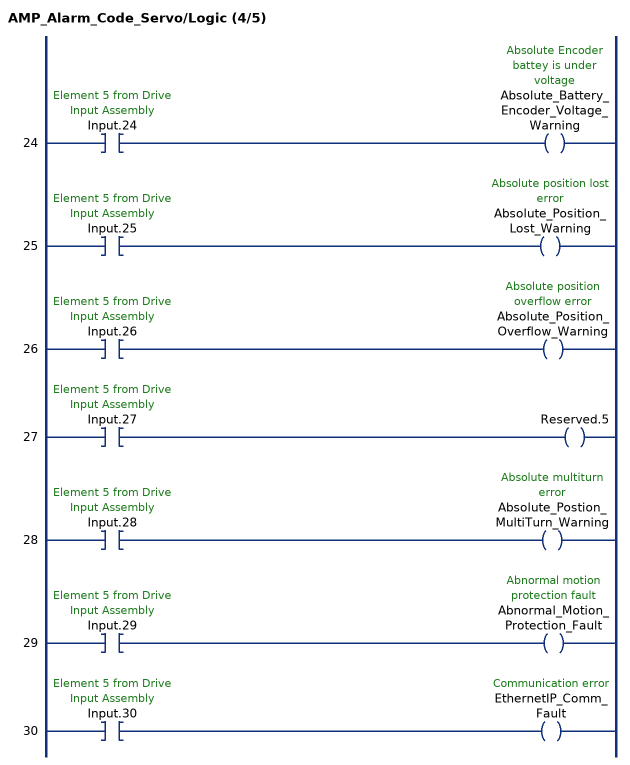
   24: XIC(Input.24)OTE(Absolute_Battery_Encoder_Voltage_Warning);
   25: XIC(Input.25)OTE(Absolute_Position_Lost_Warning);
   26: XIC(Input.26)OTE(Absolute_Position_Overflow_Warning);
   27: XIC(Input.27)OTE(Reserved.5);
   28: XIC(Input.28)OTE(Absolute_Postion_MultiTurn_Warning);
   29: XIC(Input.29)OTE(Abnormal_Motion_Protection_Fault);
   30: XIC(Input.30)OTE(EthernetIP_Comm_Fault);
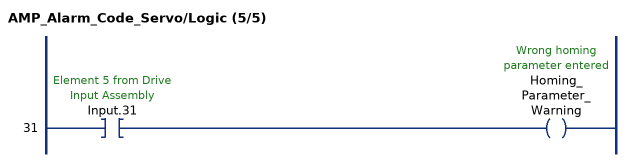
   31: XIC(Input.31)OTE(Homing_Parameter_Warning);
END_ROUTINE
END_ADD_ON_INSTRUCTION

ADD_ON_INSTRUCTION AMP_Alarm_Reset   (* revision 1.0 *)
// Applied Motion - Alarm Reset - AOI
// Help:
// The Alarm Reset AOI is used to reset Drive Fault and clear Alarm Code (if possible). Figure 1 shows a preview of an instance of the AOI.
VAR_IN_OUT
   Input : DINT[14]; {required}   // Drive Input Assembly
   Output : DINT[16]; {required}   // Drive Output Assembly
        [0]   // Command Word
        [10]   // Data/Register 1
        [11]   // Data/Register 2
        [1]   // Jog Speed (0.25 rev/min)
        [2]   // Jog Acceleration (10 rev/s/s)
        [3]   // Jog Deceleration (10 rev/s/s)
        [4]   // Point-to-Point Velocity (0.25 rev/min)
        [5]   // Point-to-Point Acceleration (10 rev/s/s)
        [6]   // Point-to-Point Deceleration (10 rev/s/s)
        [7]   // Point-to-Point Distance (Motor steps)
        [9]   // (2x ASCII Letters in 16 lower word)
END_VAR
VAR_INPUT
   RPI : DINT := 100; {visible}   // Drive Connection Request Packet Interval (milliseconds)
   Reset : BOOL; {required}   // Reset the Drive (on rising edge)
END_VAR
VAR_OUTPUT
   Sent : BOOL; {access Read Only, visible}   // Reset has been sent to drive
   In_Progress : BOOL; {access Read Only, visible}   // Reset in progress
   Done : BOOL; {access Read Only, visible}   // Reset completed without errors - Drive is not faulted
   Error : BOOL; {access Read Only, visible}   // Reset failed - Not Used
   State : DINT := 10; {access None}   // Internal state of progress
END_VAR
VAR
   Loc_StatusCode : AMP_Status_Word;
   Loc_CommandOff_Timer : TIMER;   // Timer to make sure command value was 0 before sending a new command
   Loc_CommandOn_Timer : TIMER;   // Timer to make sure command value is set long enough to be sent to servo
   Loc_Input_Assembly : AMP_Input_Assembly_v2; {access None}
   Loc_Stop_ONS : BOOL; {access None}
END_VAR

ROUTINE Logic   (* ladder *)
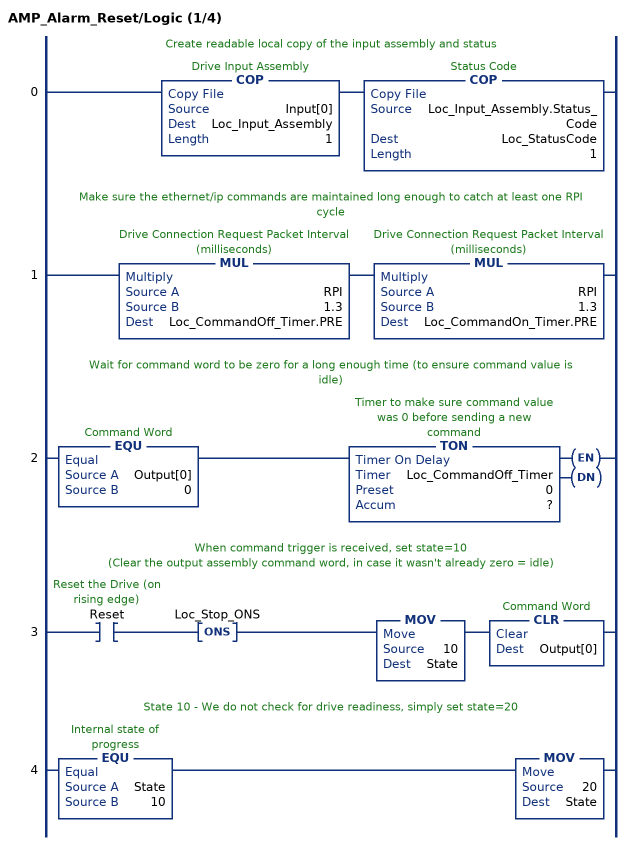
   // Create readable local copy of the input assembly and status
   0: COP(Input[0],Loc_Input_Assembly,1)COP(Loc_Input_Assembly.Status_Code,Loc_StatusCode,1);
   // Make sure the ethernet/ip commands are maintained long enough to catch at least one RPI cycle
   1: MUL(RPI,1.3,Loc_CommandOff_Timer.PRE)MUL(RPI,1.3,Loc_CommandOn_Timer.PRE);
   // Wait for command word to be zero for a long enough time (to ensure command value is idle)
   2: EQU(Output[0],0)TON(Loc_CommandOff_Timer,?,?);
   // When command trigger is received, set state=10
   // (Clear the output assembly command word, in case it wasn't already zero = idle)
   3: XIC(Reset)ONS(Loc_Stop_ONS)MOV(10,State)CLR(Output[0]);
   // State 10 - We do not check for drive readiness, simply set state=20
   4: EQU(State,10)MOV(20,State);
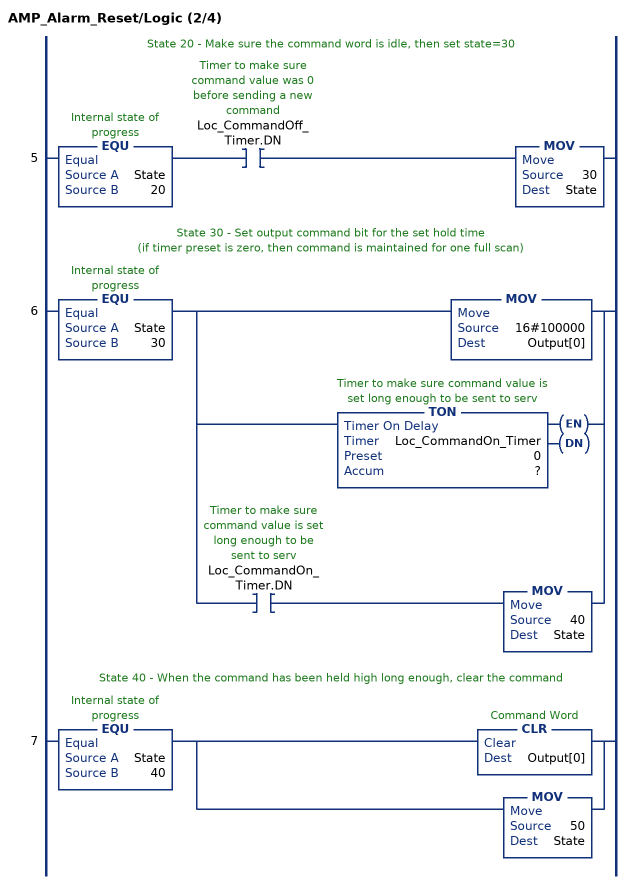
   // State 20 - Make sure the command word is idle, then set state=30
   5: EQU(State,20)XIC(Loc_CommandOff_Timer.DN)MOV(30,State);
   // State 30 - Set output command bit for the set hold time
   // (if timer preset is zero, then command is maintained for one full scan)
   6: EQU(State,30)[MOV(16#100000,Output[0]) ,TON(Loc_CommandOn_Timer,?,?) ,XIC(Loc_CommandOn_Timer.DN) MOV(40,State) ];
   // State 40 - When the command has been held high long enough, clear the command
   7: EQU(State,40)[CLR(Output[0]) ,MOV(50,State) ];
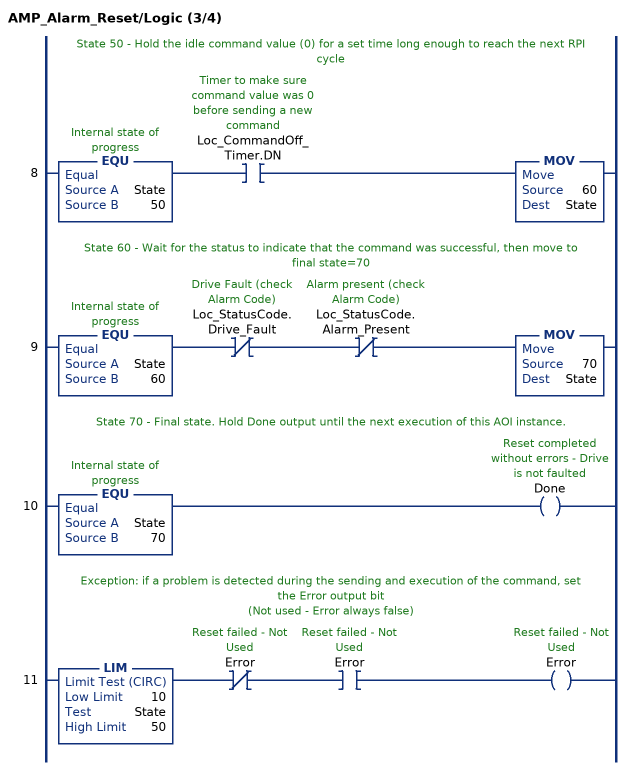
   // State 50 - Hold the idle command value (0) for a set time long enough to reach the next RPI cycle
   8: EQU(State,50)XIC(Loc_CommandOff_Timer.DN)MOV(60,State);
   // State 60 - Wait for the status to indicate that the command was successful, then move to final state=70
   9: EQU(State,60)XIO(Loc_StatusCode.Drive_Fault)XIO(Loc_StatusCode.Alarm_Present)MOV(70,State);
   // State 70 - Final state. Hold Done output until the next execution of this AOI instance.
   10: EQU(State,70)OTE(Done);
   // Exception: if a problem is detected during the sending and execution of the command, set the Error output bit
   // (Not used - Error always false)
   11: LIM(10,State,50)XIO(Error)XIC(Error)OTE(Error);
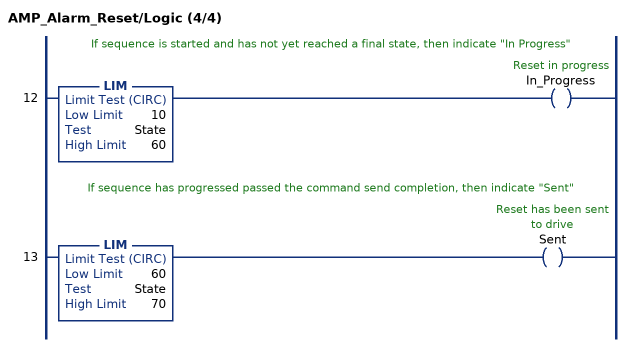
   // If sequence is started and has not yet reached a final state, then indicate "In Progress"
   12: LIM(10,State,60)OTE(In_Progress);
   // If sequence has progressed passed the command send completion, then indicate "Sent"
   13: LIM(60,State,70)OTE(Sent);
END_ROUTINE
END_ADD_ON_INSTRUCTION
